# EPICS autosave request: iocBoot/ioc1/dbSave/axs1.req
%
% BURT Request File
%
% AXIS
%

% RO $(AXS1):ActPos
$(AXS1):ActPos.DESC
$(AXS1):RqsPos
$(AXS1):RqsBkl
$(AXS1):RqsPosInc
$(AXS1):MemPos

$(AXS1):RqsPos.HOPR
$(AXS1):RqsPos.LOPR
$(AXS1):RqsPos.DRVH
$(AXS1):RqsPos.DRVL
